FUNCTION_BLOCK TestComposite
  (* Version 1.0, 2005-06-15, Goran Cengic, Chalmers *)
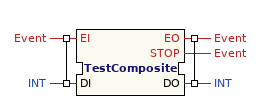
  EVENT_INPUT
    EI WITH DI;
  END_EVENT
  EVENT_OUTPUT
    EO WITH DO;
    STOP;
  END_EVENT
  VAR_INPUT
    DI : INT;
  END_VAR
  VAR_OUTPUT
    DO : INT;
  END_VAR
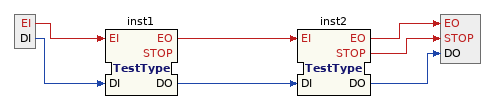
  FBS
    inst1 : TestType;
    inst2 : TestType;
  END_FBS
  EVENT_CONNECTIONS
    EI TO inst1.EI;
    inst1.EO TO inst2.EI;
    inst2.EO TO EO;
    inst2.STOP TO STOP;
  END_CONNECTIONS
  DATA_CONNECTIONS
    DI TO inst1.DI;
    inst1.DO TO inst2.DI;
    inst2.DO TO DO;
  END_CONNECTIONS
END_FUNCTION_BLOCK
